INTERFACE IMachine EXTENDS ZApplication.IUnit

END_INTERFACE

(* stored: Version 1.1.0.1
   Itf IMachine: Id {01ab74b0-26dd-4c11-be75-0f9943bd0226} *)
